FUNCTION_BLOCK FB_Modbus
VAR_INPUT
END_VAR
VAR_OUTPUT
END_VAR
VAR
	fbModbusMaster1 :		FB_ModbusMaster;
	fbModbusMaster2 :		FB_ModbusMaster;
	fbModbusSlave	:		FB_PM2200;
	fbModbusSlave1	: 		FB_TDS323PC57;
	fbModbusSlave2	: 		FB_TDS323PC57;
	fbModbusSlave3	: 		FB_TDS4339;
	istep			:		UINT;
	bStart			:		BOOL;
	
	arrData			:		ARRAY [0..255] OF BYTE := [1,3,12,16#00,16#01,16#01,16#02,16#03,16#01,16#01,16#01,16#01,16#01,16#01,16#01,3,5] ;
	fbex			:		FB_ExcitationPulseModulation;
	tonMeo			:		TON;
	btest			:		BOOL;
	
END_VAR

CASE istep OF
	0: //Trigger
		IF bStart THEN
			bStart := FALSE;
			istep := 10;
		END_IF
		
	10: //Init
		fbModbusSlave.UnitID := 1;
		fbModbusSlave.FirstCycle();
		
		fbModbusSlave1.UnitID := 1;
		fbModbusSlave1.FirstCycle();
		fbModbusSlave2.UnitID := 2;
		fbModbusSlave2.FirstCycle();
		fbModbusSlave3.UnitID := 3;
		fbModbusSlave3.FirstCycle();
		
		fbModbusMaster1.FirstCycle();
		fbModbusMaster1.Init();
		fbModbusMaster1.RegisterSlave(fbModbusSlave);
//		fbModbusMaster.RegisterSlave(fbModbusTemp);
		fbModbusMaster1.Timeout := 1000;
		
		fbModbusMaster2.FirstCycle();
		fbModbusMaster2.Init();
		fbModbusMaster2.RegisterSlave(fbModbusSlave1);
//		fbModbusMaster2.RegisterSlave(fbModbusSlave2);
//		fbModbusMaster2.RegisterSlave(fbModbusSlave3);
		fbModbusMaster2.Timeout := 1000;
		
		istep := 20;
		
	20: //Running
		IF (*fbModbusMaster1.Run()*) fbModbusMaster2.Run() THEN
			istep := 30;
		END_IF
		
	30: //Stopped
		
END_CASE

//fbModbusMaster1();
fbModbusMaster2();

fbModbusSlave.Convert(0, ADR(arrData));
fbModbusSlave1.Convert(0, ADR(arrData));
fbModbusSlave3.Convert(0, ADR(arrData));

fbex();
tonMeo(IN := NOT tonMeo.Q, PT:= T#2S);
IF btest THEN
	fbex.Increase();
END_IF

END_FUNCTION_BLOCK

(* stored: Version 1.1.0.1, ProductVersion 3.1.4024.12
   POU FB_Modbus: Id {4de26dcb-924e-4db1-99fa-8b07600b5850}, SpecialFunc None *)
